(* CoDeSys 2.3.9.35 project: Exercício 12 - Lista de ST - Testando.pro *)
(* Author: Altus *)
(* Libraries: DU35x.lib 7.7.11 15:59:13, Navigation.lib 15.7.11 10:06:00, SysLibTargetVisu.lib 26.11.08 09:53:28, Standard.lib 26.11.08 09:46:20, Iecsfc.lib 26.11.08 09:46:14, SYSLIBCALLBACK.LIB 26.11.08 09:53:30 *)

(* PLC configuration (modules and I/O channels)
Configuração do CP [Root] node -1, in %IB0 out %QB0
  Comunicação [Comunica] node 0, in %IB0 out %QB0
    COM1 [COM1] node 0, in %IB0 out %QB0 {BaudRate = 115200; Paridade = Sem Paridade; StopBits = 1 Stop Bit; Modem = Sem RTS/CTS; Delay = 5}
      MToolIEC [Codesys] node 0, in %IB0 out %QB0
    COM2 [COM2] node 1, in %IB0 out %QB0 {BaudRate = 115200; Paridade = Sem Paridade; StopBits = 1 Stop Bit; Modem = Sem RTS/CTS; Delay = 5}
      Desabilitada [Desabilitado485] node 0, in %IB0 out %QB0
  Barramento [Barramento] node 1, in %IB0 out %QB0
    Entradas [Entradas] node 0, in %IB0 out %QB0
      Entradas Digitais 0 [Entradas0] node 0, in %IW0 out %QB0
        I00 AT %IX0.0 [BitInput] I0.0
        I01 AT %IX0.1 [BitInput] I0.1
        I02 AT %IX0.2 [BitInput] I0.2
        I03 AT %IX0.3 [BitInput] I0.3
        I04 AT %IX0.4 [BitInput] I0.4
        I05 AT %IX0.5 [BitInput] I0.5
        I06 AT %IX0.6 [BitInput] I0.6
        I07 AT %IX0.7 [BitInput] I0.7
        I08 AT %IX0.8 [BitInput] I0.8
      Entradas Digitais 1 [Entradas1] node 0, in %IW1 out %QB0
        I10 AT %IX1.0 [BitInput] I1.0
        I11 AT %IX1.1 [BitInput] I1.1
        I12 AT %IX1.2 [BitInput] I1.2
        I13 AT %IX1.3 [BitInput] I1.3
        I14 AT %IX1.4 [BitInput] I1.4
        I15 AT %IX1.5 [BitInput] I1.5
        I16 AT %IX1.6 [BitInput] I1.6
        I17 AT %IX1.7 [BitInput] I1.7
        I18 AT %IX1.8 [BitInput] I1.8
      Entradas Digitais 2 [Entradas2] node 0, in %IW2 out %QB0
        I20 AT %IX2.0 [BitInput] I2.0
        I21 AT %IX2.1 [BitInput] I2.1
      Entradas Analógicas [EntradaAnalogica] node 0, in %IW4 out %QB0
        AI0 AT %IW4 [WordInput] AI0 {TipoAnalogica = Channel Disable; FiltroAnalogica = Filter 0 - AI=2ms  / AV=90ms; FundoEscala = 0}
        AI1 AT %IW5 [WordInput] AI1 {TipoAnalogica = Channel Disable; FiltroAnalogica = Filter 0 - AI=2ms  / AV=90ms; FundoEscala = 0}
        AI2 AT %IW6 [WordInput] AI2 {TipoAnalogica = Channel Disable; FiltroAnalogica = Filter 0 - AI=2ms  / AV=90ms; FundoEscala = 0}
        AI3 AT %IW7 [WordInput] AI3 {TipoAnalogica = Channel Disable; FiltroAnalogica = Filter 0 - AI=2ms  / AV=90ms; FundoEscala = 0}
      Entradas Rápidas [EntradasRapidas] node 1, in %IB16 out %QB0
        Bloco 0 [Bloco0] node 0, in %IB16 out %QB0
          Desabilitado [DesabilitadoBloco0] node 0, in %IB16 out %QB0
        Bloco 1 [Bloco1] node 1, in %IB16 out %QB0
          Desabilitado [DesabilitadoBloco1] node 0, in %IB16 out %QB0
        Entrada Configuravél Bloco 0 [EntradaConfiBloco0] node 2, in %IB16 out %QB0
          Contador 0 [EntradaConfContador0] node 0, in %IB16 out %QB0 {EntradaConfiguravelContador = Disable}
        Entrada Configuravél Bloco 1 [EntradaConfiBloco1] node 3, in %IB16 out %QB0
          Contador 2 [EntradaConfContador2] node 0, in %IB16 out %QB0 {EntradaConfiguravelContador = Disable}
    Saídas [Saidas] node 1, in %IB13 out %QB0
      Saídas Digitais 0 [Saidas0] node 0, in %IW0 out %QW0
        Q00 AT %QX0.0 [BitOutput] Q0.0
        Q01 AT %QX0.1 [BitOutput] Q0.1
        Q02 AT %QX0.2 [BitOutput] Q0.2
        Q03 AT %QX0.3 [BitOutput] Q0.3
        Q04 AT %QX0.4 [BitOutput] Q0.4
        Q05 AT %QX0.5 [BitOutput] Q0.5
        Q06 AT %QX0.6 [BitOutput] Q0.6
        Q07 AT %QX0.7 [BitOutput] Q0.7
      Saídas Digitais 1 [Saidas1] node 0, in %IW0 out %QW1
        Q10 AT %QX1.0 [BitOutput] Q1.0
        Q11 AT %QX1.1 [BitOutput] Q1.1
        Q12 AT %QX1.2 [BitOutput] Q1.2
        Q13 AT %QX1.3 [BitOutput] Q1.3
        Q14 AT %QX1.4 [BitOutput] Q1.4
        Q15 AT %QX1.5 [BitOutput] Q1.5
        Q16 AT %QX1.6 [BitOutput] Q1.6
        Q17 AT %QX1.7 [BitOutput] Q1.7
      Saídas Analógicas [SaidaAnalogica] node 0, in %IW0 out %QW3
        AO0 AT %QW3 [WordOutput] AO0 {TipoAnalogica = Channel Disable; FundoEscala = 0}
        AO1 AT %QW4 [WordOutput] AO1 {TipoAnalogica = Channel Disable; FundoEscala = 0}
      Saídas Rápidas [SaidasRapidas] node 1, in %IB0 out %QB10
        Saída Rápida 0 Desabilitada [DesabilitadoF0] node 0, in %IB0 out %QB10
        Saída Rápida 1 Desabilitada [DesabilitadoF1] node 1, in %IB0 out %QB10
      Saídas Comum de Contador [SaidasContador] node 2, in %IB0 out %QB10
        Saída do Bloco 0 Desabilitada [DesabilitadoSaidaBloco0] node 0, in %IB0 out %QB10
        Saída do Bloco 1 Desabilitada [DesabilitadoSaidaBloco1] node 1, in %IB0 out %QB10
  Eventos Externos [Eventos] node 2, in %IB13 out %QB6
    Evento Temporizado [TimerEvent] node 0, in %IB13 out %QB6 {Intervalo = 10}
*)

(* Task configuration *)
TASK PRINCIPAL (PRIORITY := 1, INTERVAL := T#1ms);
	PLC_PRG();
END_TASK
TASK NAVIGATION (PRIORITY := 1, INTERVAL := T#20ms);
	NAVEGA();
END_TASK
TASK VISUALIZATION (PRIORITY := 1, INTERVAL := T#500ms);
	MAINTARGETVISU_PAINT_CODE
END_TASK
TASK KEYBOARD_USAGE (PRIORITY := 1, INTERVAL := T#20ms);
	MAINTARGETVISU_INPUT_CODE
END_TASK

(* Data type *)
TYPE TANQUE :
	STRUCT
		LSH: BOOL;
		LSL: BOOL;
		CONCENTRACAO: REAL;
		NIVEL_MIN: INT;
		NIVEL_MAX: INT;
		ACION_BOMBA: INT;
	END_STRUCT
END_TYPE

(* POU PLC_PRG, ST *)
(*Desenvolver um sistema de gerenciamento de uma bomba de circulação de produto químico, em três tanques.

Existe um LSH (sensor de nível alto) e um LSL (sensor de nível baixo) para cada tanque. 6VAR

Para ligar a bomba (K2), nenhum dos tanques deve estar com o nível alto e o operador deve dar partida por um botão B1, podendo desligá-la pelo botão B2. 
Se o nível dentro de um dos tanques subir ao limite superior, a bomba desliga. 

Se o nível de um dos tanques atingir o limite mínimo, e nenhum dos outros tanques estiver no limite máximo, deve ser ligada a bomba K2 
e ligada a saída de alarme visual e sonoro (K1), ficando esse alarme ativo por 5 segundos . 

Crie uma estrutura para de dados para os tanques, contendo uma variável de medição do nível de concentração do produto (REAL) e duas 
variáveis de contagem (INT) dos eventos de nível máximo atingido, nível mínimo atingido (ambos de cada tanque), e de acionamentos da bomba (do sistema), 
crie um array contendo as estruturas de dados dos três tanques. 

A leitura de concentração para os três tanques é feita por sensores/transmissores analógicos (AT) que utilizam uma única entrada analógica (valor de 0,00UI 
a 50,00UI, fundo de escala 10.000) selecionada a cada 5 segundos para a leitura de cada tanque e respectiva atualização do dado no array de tanques 
(intervalo de 5s, mede tanque 1, intervalo de 5s, mede tanque 2, intervalo de 5s, mede tanque 3, e assim sucessivamente). 

Exibir na tela principal da IHM o status da bomba, do alarme e da medição atualizada dos três tanques), em uma segunda tela, exibir os contadores de eventos 
atualizados dos três tanques. Ao ser reiniciado o CLP, todas as variáveis retornam ao valor inicial "zero".
*)

PROGRAM PLC_PRG
VAR
	TANQUES: ARRAY[1..3] OF TANQUE;
	AN AT %IW4: WORD;
	T1: TON;
	T2: TON;
	M: BOOL := TRUE;
	INDEX_SENSOR: INT := 1;
	B1 AT %IX0.0: BOOL;
	B2 AT %IX0.1: BOOL;
	K2 AT %QX1.0: BOOL;
	ALARM: BOOL;
END_VAR
T1(IN := NOT M, PT := T#5s);
T2(IN := ALARM, PT := T#5s);

IF T2.Q THEN
	ALARM := FALSE;
END_IF

IF T1.Q THEN
	M := TRUE;
	TANQUES[INDEX_SENSOR].CONCENTRACAO := WORD_TO_REAL(AN) * 0.05;
	IF INDEX_SENSOR = 3 THEN
		INDEX_SENSOR := 1;
	ELSE
		INDEX_SENSOR := INDEX_SENSOR + 1;
	END_IF
ELSIF M THEN
	M := FALSE;
END_IF

IF B2 OR TANQUES[1].LSH OR TANQUES[2].LSH OR TANQUES[3].LSH THEN
	IF TANQUES[1].LSH THEN
		TANQUES[1].NIVEL_MAX := TANQUES[1].NIVEL_MAX + 1;
	ELSIF TANQUES[2].LSH THEN
		TANQUES[2].NIVEL_MAX := TANQUES[2].NIVEL_MAX + 1;
	ELSIF TANQUES[3].LSH THEN
		TANQUES[3].NIVEL_MAX := TANQUES[3].NIVEL_MAX + 1;
	END_IF
	(*CASE TRUE OF
		TANQUES[1].LSH:
			TANQUES[1].NIVEL_MAX := TANQUES[1].NIVEL_MAX + 1;
		TANQUES[2].LSH:
			TANQUES[2].NIVEL_MAX := TANQUES[2].NIVEL_MAX + 1;
		TANQUES[3].LSH:
			TANQUES[3].NIVEL_MAX := TANQUES[3].NIVEL_MAX + 1;
	END_CASE*)
	K2 := FALSE;
ELSIF B1 OR TANQUES[1].LSL OR TANQUES[2].LSL OR TANQUES[3].LSL THEN
	IF TANQUES[1].LSL THEN
		TANQUES[1].ACION_BOMBA := TANQUES[1].ACION_BOMBA + 1;
		TANQUES[1].NIVEL_MIN := TANQUES[1].NIVEL_MIN + 1;
		ALARM := TRUE;
	ELSIF TANQUES[2].LSL THEN
		TANQUES[2].ACION_BOMBA := TANQUES[2].ACION_BOMBA + 1;
		TANQUES[2].NIVEL_MIN := TANQUES[2].NIVEL_MIN + 1;
		ALARM := TRUE;
	ELSIF TANQUES[3].LSL THEN
		TANQUES[3].ACION_BOMBA := TANQUES[3].ACION_BOMBA + 1;
		TANQUES[3].NIVEL_MIN := TANQUES[3].NIVEL_MIN + 1;
		ALARM := TRUE;
	END_IF
	(*CASE TRUE OF
		TANQUES[1].LSL:
			TANQUES[1].ACION_BOMBA := TANQUES[1].ACION_BOMBA + 1;
			TANQUES[1].NIVEL_MIN := TANQUES[1].NIVEL_MIN + 1;
			ALARM := TRUE;
		TANQUES[2].LSL:
			TANQUES[2].ACION_BOMBA := TANQUES[2].ACION_BOMBA + 1;
			TANQUES[2].NIVEL_MIN := TANQUES[2].NIVEL_MIN + 1;
			ALARM := TRUE;
		TANQUES[3].LSL:
			TANQUES[3].ACION_BOMBA := TANQUES[3].ACION_BOMBA + 1;
			TANQUES[3].NIVEL_MIN := TANQUES[3].NIVEL_MIN + 1;
			ALARM := TRUE;
	END_CASE*)
	K2 := TRUE;
END_IF
END_PROGRAM

(* POU NAVEGA, ST *)
PROGRAM NAVEGA
VAR
	ControleTelas : NAVIGATION;
	ListaTelas 	: ARRAY [0..30] OF STRING(10);
END_VAR
(* Adiciona a tela MAIN como tela principal *)
ListaTelas[0] := 'MAIN';

(* Ativa o controle automático de navegação somente pelo teclado *)
ControleTelas(ENABLE_UPDW := FALSE, VISU_LIST := ListaTelas, UP := FALSE , DOWN := FALSE);
END_PROGRAM
